TYPE E_Destination :
(
	StackerA,
	StackerB,
	StackerC,
	Garbage,
	MAX_E_Destination
);
END_TYPE

(* stored: Version 1.1.0.1, ProductVersion 3.1.0.24
   DUT E_Destination: Id {68cd0b97-d771-42fd-a06d-0b95e803d339} *)
